FUNCTION_BLOCK JsonDeserializerObjectForwardEnumerator_TestSuite EXTENDS TcUnit.FB_TestSuite
VAR
END_VAR

TestIsValidAtStart();
TestIsNotValidAfterParentReset();
TestMoveNextReturnsFalseAtTheEnd();
TestMoveNextReturnsTrueSingleItem();
TestMoveNextReturnsFalseWhenEmpty();
TestMoveNextReturnsTrueMultipleItems();
TestEnumerateThroughKeys();

METHOD PRIVATE TestEnumerateThroughKeys
VAR
	jsonDeserializer : JsonDeserializer;
	enumerator : I_DeserializerObjectForwardEnumerator;
    json : STRING := '{"key1":"value1", "key2":"value2", "key3":"value3"}';
	out1, out2, out3 : STRING;
	expected1 : STRING := 'key1';
	expected2 : STRING := 'key2';
	expected3 : STRING := 'key3';
	result : BOOL;
END_VAR
TEST('TestEnumerateThroughKeys');

jsonDeserializer.TryLoad(json);
enumerator := jsonDeserializer.GetObjectEnumerator();

enumerator.MoveNext();
out1 := enumerator.Key;

enumerator.MoveNext();
out2 := enumerator.Key;

enumerator.MoveNext();
out3 := enumerator.Key;

enumerator.Dispose();

AssertEquals(
	Expected := expected1,
	Actual := out1,
	Message := 'Did not produce the expected result'
);

AssertEquals(
	Expected := expected2,
	Actual := out2,
	Message := 'Did not produce the expected result'
);

AssertEquals(
	Expected := expected3,
	Actual := out3,
	Message := 'Did not produce the expected result'
);
	
TEST_FINISHED();
END_METHOD

METHOD PRIVATE TestIsNotValidAfterParentReset
VAR
	jsonDeserializer : JsonDeserializer;
	enumerator : I_DeserializerObjectForwardEnumerator;
	result : BOOL;
END_VAR
TEST('TestIsNotValidAfterParentReset');

enumerator := jsonDeserializer.GetObjectEnumerator();

jsonDeserializer.Reset();
result := enumerator.IsValid;

enumerator.Dispose();

AssertFalse(
	Condition := result,
	Message := 'IsValid incorrectly returned true after parent was reset'
);

TEST_FINISHED();
END_METHOD

METHOD PRIVATE TestIsValidAtStart
VAR
	jsonDeserializer : JsonDeserializer;
	enumerator : I_DeserializerObjectForwardEnumerator;
	result : BOOL;
END_VAR
TEST('TestIsValidAtStart');

enumerator := jsonDeserializer.GetObjectEnumerator();

result := enumerator.IsValid;
enumerator.Dispose();

AssertTrue(
	Condition := result,
	Message := 'IsValid returned false'
);

TEST_FINISHED();
END_METHOD

METHOD PRIVATE TestMoveNextReturnsFalseAtTheEnd
VAR
	jsonDeserializer : JsonDeserializer;
	enumerator : I_DeserializerObjectForwardEnumerator;
    json : STRING := '{"key1":"value1"}';
	result : BOOL;
END_VAR
TEST('CheckMoveNextReturnsFalseAtTheEnd');

jsonDeserializer.TryLoad(json);
enumerator := jsonDeserializer.GetObjectEnumerator();

enumerator.MoveNext();
result := enumerator.MoveNext();

enumerator.Dispose();

AssertFalse(result,
    'MoveNext did not correctly signal the end of the enumeration');
	
TEST_FINISHED();
END_METHOD

METHOD PRIVATE TestMoveNextReturnsFalseWhenEmpty
VAR
	jsonDeserializer : JsonDeserializer;
	enumerator : I_DeserializerObjectForwardEnumerator;
    json : STRING := '{}';
	result : BOOL;
END_VAR
TEST('CheckMoveNextReturnsFalseWhenEmpty');

jsonDeserializer.TryLoad(json);
enumerator := jsonDeserializer.GetObjectEnumerator();

result := enumerator.MoveNext();

enumerator.Dispose();

AssertFalse(result,
    'MoveNext did not correctly signal an empty array');
	
TEST_FINISHED();
END_METHOD

METHOD PRIVATE TestMoveNextReturnsTrueMultipleItems
VAR
	jsonDeserializer : JsonDeserializer;
	enumerator : I_DeserializerObjectForwardEnumerator;
    json : STRING := '{"key1":"value1", "key2":"value2"}';
	result : BOOL;
END_VAR
TEST('CheckMoveNextReturnsTrueMultipleItems');

jsonDeserializer.TryLoad(json);
enumerator := jsonDeserializer.GetObjectEnumerator();

enumerator.MoveNext();
result := enumerator.MoveNext();

enumerator.Dispose();

AssertTrue(
	Condition := result,
	Message := 'MoveNext did not correctly signal there were more items to follow'
);
	
TEST_FINISHED();
END_METHOD

METHOD PRIVATE TestMoveNextReturnsTrueSingleItem
VAR
	jsonDeserializer : JsonDeserializer;
	enumerator : I_DeserializerObjectForwardEnumerator;
    json : STRING := '{"key1":"value1"}';
	result : BOOL;
END_VAR
TEST('CheckMoveNextReturnsTrueSingleItem');

jsonDeserializer.TryLoad(json);
enumerator := jsonDeserializer.GetObjectEnumerator();

result := enumerator.MoveNext();

enumerator.Dispose();

AssertTrue(
	Condition := result,
	Message := 'MoveNext did not correctly signal there were more items to follow, i.e. the first item'
);
	
TEST_FINISHED();
END_METHOD

END_FUNCTION_BLOCK

(* stored: Version 1.1.0.1, ProductVersion 3.1.4024.12
   POU JsonDeserializerObjectForwardEnumerator_TestSuite: Id {9df7fd9c-1b17-45ef-bc71-b2204df2de81}, SpecialFunc None
   Method TestEnumerateThroughKeys: Id {2119cc28-70e0-4b53-99e2-519c940091a4}
   Method TestIsNotValidAfterParentReset: Id {301560c1-670d-4067-a959-1b45c0721292}
   Method TestIsValidAtStart: Id {e56f0dba-648e-4cad-ae1c-d4a58160e91f}
   Method TestMoveNextReturnsFalseAtTheEnd: Id {5f5163d9-ff08-49e9-94e8-ed56df5f16ca}
   Method TestMoveNextReturnsFalseWhenEmpty: Id {f6eb5634-188b-4ab4-b874-e36fc78b94f0}
   Method TestMoveNextReturnsTrueMultipleItems: Id {9def64da-4a95-44bf-bd1f-ef3f29903634}
   Method TestMoveNextReturnsTrueSingleItem: Id {177e6b97-c760-4dd4-8273-5ec8f3b9a363} *)
